IF Main.Errors.InMoldDryingErrors.TopMoldB.HeatingZone[2].PT100_TemperatureAboveMaximum THEN 
Topmold_B_heating_zone_2_temperature_above_250_degree_heating_element_switched_off.Raise(Main.timestampNanoseconds); 
END_IF 

IF Main.Errors.InMoldDryingErrors.TopMoldB.HeatingZone[2].PT100_TemperatureTooHighWarn THEN 
Topmold_B_heating_zone_2_temperature_above_230_degree.Raise(Main.timestampNanoseconds); 
END_IF 

IF Main.Errors.InMoldDryingErrors.TopMoldB.HeatingZone[3].PT100_ConnectorNotConnected THEN 
Topmold_B_heating_Zone_3_connector_not_connected.Raise(Main.timestampNanoseconds); 
END_IF 

IF Main.Errors.InMoldDryingErrors.TopMoldB.HeatingZone[3].PT100_HasWrongPosition THEN 
Topmold_B_heating_Zone_3_PT100_wrong_position.Raise(Main.timestampNanoseconds); 
END_IF 

IF Main.Errors.InMoldDryingErrors.TopMoldB.HeatingZone[3].PT100_Loose THEN 
Topmold_B_heating_Zone_3_PT100_loose.Raise(Main.timestampNanoseconds); 
END_IF 

IF Main.Errors.InMoldDryingErrors.TopMoldB.HeatingZone[3].PT100_NotInserted THEN 
Topmold_B_heating_Zone_3_PT100_not_inserted.Raise(Main.timestampNanoseconds); 
END_IF 

IF Main.Errors.InMoldDryingErrors.TopMoldB.HeatingZone[3].PT100_TempAboveSetpoint THEN 
Topmold_B_heating_Zone_3_Temperature_above_setpoint.Raise(Main.timestampNanoseconds); 
END_IF 

IF Main.Errors.InMoldDryingErrors.TopMoldB.HeatingZone[3].PT100_TempBelowSetpoint THEN 
Topmold_B_heating_Zone_3_Temperature_below_setpoint.Raise(Main.timestampNanoseconds); 
END_IF 

IF Main.Errors.InMoldDryingErrors.TopMoldB.HeatingZone[3].PT100_WireBreak THEN 
Topmold_B_heating_Zone_3_PT100_wirebreak.Raise(Main.timestampNanoseconds); 
END_IF 

IF Main.Errors.InMoldDryingErrors.TopMoldB.HeatingZone[3].Thermal THEN 
Topmold_B_heating_Zone_3_Thermal.Raise(Main.timestampNanoseconds); 
END_IF 

IF Main.Errors.InMoldDryingErrors.TopMoldB.HeatingZone[3].PT100_TemperatureAboveMaximum THEN 
Topmold_B_heating_zone_3_temperature_above_250_degree_heating_element_switched_off.Raise(Main.timestampNanoseconds); 
END_IF 

IF Main.Errors.InMoldDryingErrors.TopMoldB.HeatingZone[3].PT100_TemperatureTooHighWarn THEN 
Topmold_B_heating_zone_3_temperature_above_230_degree.Raise(Main.timestampNanoseconds); 
END_IF 

IF Main.Errors.InMoldDryingErrors.TopMoldB.HeatingZone[4].PT100_ConnectorNotConnected THEN 
Topmold_B_heating_Zone_4_connector_not_connected.Raise(Main.timestampNanoseconds); 
END_IF 

IF Main.Errors.InMoldDryingErrors.TopMoldB.HeatingZone[4].PT100_HasWrongPosition THEN 
Topmold_B_heating_Zone_4_PT100_wrong_position.Raise(Main.timestampNanoseconds); 
END_IF 

IF Main.Errors.InMoldDryingErrors.TopMoldB.HeatingZone[4].PT100_Loose THEN 
Topmold_B_heating_Zone_4_PT100_loose.Raise(Main.timestampNanoseconds); 
END_IF 

IF Main.Errors.InMoldDryingErrors.TopMoldB.HeatingZone[4].PT100_NotInserted THEN 
Topmold_B_heating_Zone_4_PT100_not_inserted.Raise(Main.timestampNanoseconds); 
END_IF 

IF Main.Errors.InMoldDryingErrors.TopMoldB.HeatingZone[4].PT100_TempAboveSetpoint THEN 
Topmold_B_heating_Zone_4_Temperature_above_setpoint.Raise(Main.timestampNanoseconds); 
END_IF 

IF Main.Errors.InMoldDryingErrors.TopMoldB.HeatingZone[4].PT100_TempBelowSetpoint THEN 
Topmold_B_heating_Zone_4_Temperature_below_setpoint.Raise(Main.timestampNanoseconds); 
END_IF 

IF Main.Errors.InMoldDryingErrors.TopMoldB.HeatingZone[4].PT100_WireBreak THEN 
Topmold_B_heating_Zone_4_PT100_wirebreak.Raise(Main.timestampNanoseconds); 
END_IF 

IF Main.Errors.InMoldDryingErrors.TopMoldB.HeatingZone[4].Thermal THEN 
Topmold_B_heating_Zone_4_Thermal.Raise(Main.timestampNanoseconds); 
END_IF 

IF Main.Errors.InMoldDryingErrors.TopMoldB.HeatingZone[4].PT100_TemperatureAboveMaximum THEN 
Topmold_B_heating_zone_4_temperature_above_250_degree_heating_element_switched_off.Raise(Main.timestampNanoseconds); 
END_IF 

IF Main.Errors.InMoldDryingErrors.TopMoldB.HeatingZone[4].PT100_TemperatureTooHighWarn THEN 
Topmold_B_heating_zone_4_temperature_above_230_degree.Raise(Main.timestampNanoseconds); 
END_IF 

IF Main.Errors.InMoldDryingErrors.TopMoldB.HeatingZone[5].PT100_ConnectorNotConnected THEN 
Topmold_B_heating_Zone_5_connector_not_connected.Raise(Main.timestampNanoseconds); 
END_IF 

IF Main.Errors.InMoldDryingErrors.TopMoldB.HeatingZone[5].PT100_HasWrongPosition THEN 
Topmold_B_heating_Zone_5_PT100_wrong_position.Raise(Main.timestampNanoseconds); 
END_IF 

IF Main.Errors.InMoldDryingErrors.TopMoldB.HeatingZone[5].PT100_Loose THEN 
Topmold_B_heating_Zone_5_PT100_loose.Raise(Main.timestampNanoseconds); 
END_IF 

IF Main.Errors.InMoldDryingErrors.TopMoldB.HeatingZone[5].PT100_NotInserted THEN 
Topmold_B_heating_Zone_5_PT100_not_inserted.Raise(Main.timestampNanoseconds); 
END_IF 

IF Main.Errors.InMoldDryingErrors.TopMoldB.HeatingZone[5].PT100_TempAboveSetpoint THEN 
Topmold_B_heating_Zone_5_Temperature_above_setpoint.Raise(Main.timestampNanoseconds); 
END_IF 

IF Main.Errors.InMoldDryingErrors.TopMoldB.HeatingZone[5].PT100_TempBelowSetpoint THEN 
Topmold_B_heating_Zone_5_Temperature_below_setpoint.Raise(Main.timestampNanoseconds); 
END_IF 

IF Main.Errors.InMoldDryingErrors.TopMoldB.HeatingZone[5].PT100_WireBreak THEN 
Topmold_B_heating_Zone_5_PT100_wirebreak.Raise(Main.timestampNanoseconds); 
END_IF 

IF Main.Errors.InMoldDryingErrors.TopMoldB.HeatingZone[5].Thermal THEN 
Topmold_B_heating_Zone_5_Thermal.Raise(Main.timestampNanoseconds); 
END_IF 

IF Main.Errors.InMoldDryingErrors.TopMoldB.HeatingZone[5].PT100_TemperatureAboveMaximum THEN 
Topmold_B_heating_zone_5_temperature_above_250_degree_heating_element_switched_off.Raise(Main.timestampNanoseconds); 
END_IF 

IF Main.Errors.InMoldDryingErrors.TopMoldB.HeatingZone[5].PT100_TemperatureTooHighWarn THEN 
Topmold_B_heating_zone_5_temperature_above_230_degree.Raise(Main.timestampNanoseconds); 
END_IF 

IF Main.Errors.InMoldDryingErrors.TopMoldB.HeatingZone[6].PT100_ConnectorNotConnected THEN 
Topmold_B_heating_Zone_6_connector_not_connected.Raise(Main.timestampNanoseconds); 
END_IF 

IF Main.Errors.InMoldDryingErrors.TopMoldB.HeatingZone[6].PT100_HasWrongPosition THEN 
Topmold_B_heating_Zone_6_PT100_wrong_position.Raise(Main.timestampNanoseconds); 
END_IF 

IF Main.Errors.InMoldDryingErrors.TopMoldB.HeatingZone[6].PT100_Loose THEN 
Topmold_B_heating_Zone_6_PT100_loose.Raise(Main.timestampNanoseconds); 
END_IF 

IF Main.Errors.InMoldDryingErrors.TopMoldB.HeatingZone[6].PT100_NotInserted THEN 
Topmold_B_heating_Zone_6_PT100_not_inserted.Raise(Main.timestampNanoseconds); 
END_IF 

IF Main.Errors.InMoldDryingErrors.TopMoldB.HeatingZone[6].PT100_TempAboveSetpoint THEN 
Topmold_B_heating_Zone_6_Temperature_above_setpoint.Raise(Main.timestampNanoseconds); 
END_IF 

IF Main.Errors.InMoldDryingErrors.TopMoldB.HeatingZone[6].PT100_TempBelowSetpoint THEN 
Topmold_B_heating_Zone_6_Temperature_below_setpoint.Raise(Main.timestampNanoseconds); 
END_IF 

IF Main.Errors.InMoldDryingErrors.TopMoldB.HeatingZone[6].PT100_WireBreak THEN 
Topmold_B_heating_Zone_6_PT100_wirebreak.Raise(Main.timestampNanoseconds); 
END_IF 

IF Main.Errors.InMoldDryingErrors.TopMoldB.HeatingZone[6].Thermal THEN 
Topmold_B_heating_Zone_6_Thermal.Raise(Main.timestampNanoseconds); 
END_IF 

IF Main.Errors.InMoldDryingErrors.TopMoldB.HeatingZone[6].PT100_TemperatureAboveMaximum THEN 
Topmold_B_heating_zone_6_temperature_above_250_degree_heating_element_switched_off.Raise(Main.timestampNanoseconds); 
END_IF 

IF Main.Errors.InMoldDryingErrors.TopMoldB.HeatingZone[6].PT100_TemperatureTooHighWarn THEN 
Topmold_B_heating_zone_6_temperature_above_230_degree.Raise(Main.timestampNanoseconds); 
END_IF 

IF Main.Errors.InMoldDryingErrors.TopMoldB.Hydraulic.BallufError THEN 
Bottom_mold_B_error_on_balluf.Raise(Main.timestampNanoseconds); 
END_IF 

IF Main.Errors.InMoldDryingErrors.TopMoldB.Hydraulic.IsMovingWithoutActivation THEN 
Bottom_mold_B_is_moving_without_activation.Raise(Main.timestampNanoseconds); 
END_IF 

IF FALSE THEN 
Top_mold_B_Bot_side_pressure_too_high.Raise(Main.timestampNanoseconds); 
END_IF 

IF FALSE THEN 
Top_mold_B_Rot_side_pressure_too_high.Raise(Main.timestampNanoseconds); 
END_IF 

IF Main.Errors.InMoldDryingErrors.BottomMoldB.HeatingZone[1].PT100_ConnectorNotConnected THEN 
Bottom_mold_B_heating_Zone_1_connector_not_connected.Raise(Main.timestampNanoseconds); 
END_IF 

IF Main.Errors.InMoldDryingErrors.BottomMoldB.HeatingZone[1].PT100_HasWrongPosition THEN 
Bottom_mold_B_heating_Zone_1_PT100_wrong_position.Raise(Main.timestampNanoseconds); 
END_IF 

IF Main.Errors.InMoldDryingErrors.BottomMoldB.HeatingZone[1].PT100_Loose THEN 
Bottom_mold_B_heating_Zone_1_PT100_loose.Raise(Main.timestampNanoseconds); 
END_IF 

IF Main.Errors.InMoldDryingErrors.BottomMoldB.HeatingZone[1].PT100_NotInserted THEN 
Bottom_mold_B_heating_Zone_1_PT100_not_inserted.Raise(Main.timestampNanoseconds); 
END_IF 

IF Main.Errors.InMoldDryingErrors.BottomMoldB.HeatingZone[1].PT100_TempAboveSetpoint THEN 
Bottom_mold_B_heating_Zone_1_Temperature_above_setpoint.Raise(Main.timestampNanoseconds); 
END_IF 

IF Main.Errors.InMoldDryingErrors.BottomMoldB.HeatingZone[1].PT100_TempBelowSetpoint THEN 
Bottom_mold_B_heating_Zone_1_Temperature_below_setpoint.Raise(Main.timestampNanoseconds); 
END_IF 

IF Main.Errors.InMoldDryingErrors.BottomMoldB.HeatingZone[1].PT100_WireBreak THEN 
Bottom_mold_B_heating_Zone_1_PT100_wirebreak.Raise(Main.timestampNanoseconds); 
END_IF 

IF Main.Errors.InMoldDryingErrors.BottomMoldB.HeatingZone[1].Thermal THEN 
Bottom_mold_B_heating_Zone_1_Thermal.Raise(Main.timestampNanoseconds); 
END_IF 

IF Main.Errors.InMoldDryingErrors.BottomMoldB.HeatingZone[1].PT100_TemperatureAboveMaximum THEN 
Bottom_mold_B_heating_zone_1_temperature_above_250_degree_heating_element_switched_off.Raise(Main.timestampNanoseconds); 
END_IF 

IF Main.Errors.InMoldDryingErrors.BottomMoldB.HeatingZone[1].PT100_TemperatureTooHighWarn THEN 
Bottom_mold_B_heating_zone_1_temperature_above_230_degree.Raise(Main.timestampNanoseconds); 
END_IF 

IF Main.Errors.InMoldDryingErrors.BottomMoldB.HeatingZone[2].PT100_ConnectorNotConnected THEN 
Bottom_mold_B_heating_Zone_2_connector_not_connected.Raise(Main.timestampNanoseconds); 
END_IF 

IF Main.Errors.InMoldDryingErrors.BottomMoldB.HeatingZone[2].PT100_HasWrongPosition THEN 
Bottom_mold_B_heating_Zone_2_PT100_wrong_position.Raise(Main.timestampNanoseconds); 
END_IF 

IF Main.Errors.InMoldDryingErrors.BottomMoldB.HeatingZone[2].PT100_Loose THEN 
Bottom_mold_B_heating_Zone_2_PT100_loose.Raise(Main.timestampNanoseconds); 
END_IF 

IF Main.Errors.InMoldDryingErrors.BottomMoldB.HeatingZone[2].PT100_NotInserted THEN 
Bottom_mold_B_heating_Zone_2_PT100_not_inserted.Raise(Main.timestampNanoseconds); 
END_IF 

IF Main.Errors.InMoldDryingErrors.BottomMoldB.HeatingZone[2].PT100_TempAboveSetpoint THEN 
Bottom_mold_B_heating_Zone_2_Temperature_above_setpoint.Raise(Main.timestampNanoseconds); 
END_IF 

IF Main.Errors.InMoldDryingErrors.BottomMoldB.HeatingZone[2].PT100_TempBelowSetpoint THEN 
Bottom_mold_B_heating_Zone_2_Temperature_below_setpoint.Raise(Main.timestampNanoseconds); 
END_IF 

IF Main.Errors.InMoldDryingErrors.BottomMoldB.HeatingZone[2].PT100_WireBreak THEN 
Bottom_mold_B_heating_Zone_2_PT100_wirebreak.Raise(Main.timestampNanoseconds); 
END_IF 

IF Main.Errors.InMoldDryingErrors.BottomMoldB.HeatingZone[2].Thermal THEN 
Bottom_mold_B_heating_Zone_2_Thermal.Raise(Main.timestampNanoseconds); 
END_IF 

IF Main.Errors.InMoldDryingErrors.BottomMoldB.HeatingZone[2].PT100_TemperatureAboveMaximum THEN 
Bottom_mold_B_heating_zone_2_temperature_above_250_degree_heating_element_switched_off.Raise(Main.timestampNanoseconds); 
END_IF 

IF Main.Errors.InMoldDryingErrors.BottomMoldB.HeatingZone[2].PT100_TemperatureTooHighWarn THEN 
Bottom_mold_B_heating_zone_2_temperature_above_230_degree.Raise(Main.timestampNanoseconds); 
END_IF 

IF Main.Errors.InMoldDryingErrors.BottomMoldB.HeatingZone[3].PT100_ConnectorNotConnected THEN 
Bottom_mold_B_heating_Zone_3_connector_not_connected.Raise(Main.timestampNanoseconds); 
END_IF 

IF Main.Errors.InMoldDryingErrors.BottomMoldB.HeatingZone[3].PT100_HasWrongPosition THEN 
Bottom_mold_B_heating_Zone_3_PT100_wrong_position.Raise(Main.timestampNanoseconds); 
END_IF 

IF Main.Errors.InMoldDryingErrors.BottomMoldB.HeatingZone[3].PT100_Loose THEN 
Bottom_mold_B_heating_Zone_3_PT100_loose.Raise(Main.timestampNanoseconds); 
END_IF 

IF Main.Errors.InMoldDryingErrors.BottomMoldB.HeatingZone[3].PT100_NotInserted THEN 
Bottom_mold_B_heating_Zone_3_PT100_not_inserted.Raise(Main.timestampNanoseconds); 
END_IF 

IF Main.Errors.InMoldDryingErrors.BottomMoldB.HeatingZone[3].PT100_TempAboveSetpoint THEN 
Bottom_mold_B_heating_Zone_3_Temperature_above_setpoint.Raise(Main.timestampNanoseconds); 
END_IF 

IF Main.Errors.InMoldDryingErrors.BottomMoldB.HeatingZone[3].PT100_TempBelowSetpoint THEN 
Bottom_mold_B_heating_Zone_3_Temperature_below_setpoint.Raise(Main.timestampNanoseconds); 
END_IF 

IF Main.Errors.InMoldDryingErrors.BottomMoldB.HeatingZone[3].PT100_WireBreak THEN 
Bottom_mold_B_heating_Zone_3_PT100_wirebreak.Raise(Main.timestampNanoseconds); 
END_IF 

IF Main.Errors.InMoldDryingErrors.BottomMoldB.HeatingZone[3].Thermal THEN 
Bottom_mold_B_heating_Zone_3_Thermal.Raise(Main.timestampNanoseconds); 
END_IF 

IF Main.Errors.InMoldDryingErrors.BottomMoldB.HeatingZone[3].PT100_TemperatureAboveMaximum THEN 
Bottom_mold_B_heating_zone_3_temperature_above_250_degree_heating_element_switched_off.Raise(Main.timestampNanoseconds); 
END_IF 

IF Main.Errors.InMoldDryingErrors.BottomMoldB.HeatingZone[3].PT100_TemperatureTooHighWarn THEN 
Bottom_mold_B_heating_zone_3_temperature_above_230_degree.Raise(Main.timestampNanoseconds); 
END_IF 

IF Main.Errors.InMoldDryingErrors.BottomMoldB.HeatingZone[4].PT100_ConnectorNotConnected THEN 
Bottom_mold_B_heating_Zone_4_connector_not_connected.Raise(Main.timestampNanoseconds); 
END_IF 

IF Main.Errors.InMoldDryingErrors.BottomMoldB.HeatingZone[4].PT100_HasWrongPosition THEN 
Bottom_mold_B_heating_Zone_4_PT100_wrong_position.Raise(Main.timestampNanoseconds); 
END_IF 

IF Main.Errors.InMoldDryingErrors.BottomMoldB.HeatingZone[4].PT100_Loose THEN 
Bottom_mold_B_heating_Zone_4_PT100_loose.Raise(Main.timestampNanoseconds); 
END_IF 

IF Main.Errors.InMoldDryingErrors.BottomMoldB.HeatingZone[4].PT100_NotInserted THEN 
Bottom_mold_B_heating_Zone_4_PT100_not_inserted.Raise(Main.timestampNanoseconds); 
END_IF 

IF Main.Errors.InMoldDryingErrors.BottomMoldB.HeatingZone[4].PT100_TempAboveSetpoint THEN 
Bottom_mold_B_heating_Zone_4_Temperature_above_setpoint.Raise(Main.timestampNanoseconds); 
END_IF 

IF Main.Errors.InMoldDryingErrors.BottomMoldB.HeatingZone[4].PT100_TempBelowSetpoint THEN 
Bottom_mold_B_heating_Zone_4_Temperature_below_setpoint.Raise(Main.timestampNanoseconds); 
END_IF 

IF Main.Errors.InMoldDryingErrors.BottomMoldB.HeatingZone[4].PT100_WireBreak THEN 
Bottom_mold_B_heating_Zone_4_PT100_wirebreak.Raise(Main.timestampNanoseconds); 
END_IF 

IF Main.Errors.InMoldDryingErrors.BottomMoldB.HeatingZone[4].Thermal THEN 
Bottom_mold_B_heating_Zone_4_Thermal.Raise(Main.timestampNanoseconds); 
END_IF 

IF Main.Errors.InMoldDryingErrors.BottomMoldB.HeatingZone[4].PT100_TemperatureAboveMaximum THEN 
Bottom_mold_B_heating_zone_4_temperature_above_250_degree_heating_element_switched_off.Raise(Main.timestampNanoseconds); 
END_IF 

IF Main.Errors.InMoldDryingErrors.BottomMoldB.HeatingZone[4].PT100_TemperatureTooHighWarn THEN 
Bottom_mold_B_heating_zone_4_temperature_above_230_degree.Raise(Main.timestampNanoseconds); 
END_IF 

IF Main.Errors.InMoldDryingErrors.BottomMoldB.HeatingZone[5].PT100_ConnectorNotConnected THEN 
Bottom_mold_B_heating_Zone_5_connector_not_connected.Raise(Main.timestampNanoseconds); 
END_IF 

IF Main.Errors.InMoldDryingErrors.BottomMoldB.HeatingZone[5].PT100_HasWrongPosition THEN 
Bottom_mold_B_heating_Zone_5_PT100_wrong_position.Raise(Main.timestampNanoseconds); 
END_IF 

IF Main.Errors.InMoldDryingErrors.BottomMoldB.HeatingZone[5].PT100_Loose THEN 
Bottom_mold_B_heating_Zone_5_PT100_loose.Raise(Main.timestampNanoseconds); 
END_IF 

IF Main.Errors.InMoldDryingErrors.BottomMoldB.HeatingZone[5].PT100_NotInserted THEN 
Bottom_mold_B_heating_Zone_5_PT100_not_inserted.Raise(Main.timestampNanoseconds); 
END_IF 

IF Main.Errors.InMoldDryingErrors.BottomMoldB.HeatingZone[5].PT100_TempAboveSetpoint THEN 
Bottom_mold_B_heating_Zone_5_Temperature_above_setpoint.Raise(Main.timestampNanoseconds); 
END_IF 

IF Main.Errors.InMoldDryingErrors.BottomMoldB.HeatingZone[5].PT100_TempBelowSetpoint THEN 
Bottom_mold_B_heating_Zone_5_Temperature_below_setpoint.Raise(Main.timestampNanoseconds); 
END_IF 

IF Main.Errors.InMoldDryingErrors.BottomMoldB.HeatingZone[5].PT100_WireBreak THEN 
Bottom_mold_B_heating_Zone_5_PT100_wirebreak.Raise(Main.timestampNanoseconds); 
END_IF 

IF Main.Errors.InMoldDryingErrors.BottomMoldB.HeatingZone[5].Thermal THEN 
Bottom_mold_B_heating_Zone_5_Thermal.Raise(Main.timestampNanoseconds); 
END_IF 

IF Main.Errors.InMoldDryingErrors.BottomMoldB.HeatingZone[5].PT100_TemperatureAboveMaximum THEN 
Bottom_mold_B_heating_zone_5_temperature_above_250_degree_heating_element_switched_off.Raise(Main.timestampNanoseconds); 
END_IF 

IF Main.Errors.InMoldDryingErrors.BottomMoldB.HeatingZone[5].PT100_TemperatureTooHighWarn THEN 
Bottom_mold_B_heating_zone_5_temperature_above_230_degree.Raise(Main.timestampNanoseconds); 
END_IF 

IF Main.Errors.InMoldDryingErrors.BottomMoldB.HeatingZone[6].PT100_ConnectorNotConnected THEN 
Bottom_mold_B_heating_Zone_6_connector_not_connected.Raise(Main.timestampNanoseconds); 
END_IF 

IF Main.Errors.InMoldDryingErrors.BottomMoldB.HeatingZone[6].PT100_HasWrongPosition THEN 
Bottom_mold_B_heating_Zone_6_PT100_wrong_position.Raise(Main.timestampNanoseconds); 
END_IF 

IF Main.Errors.InMoldDryingErrors.BottomMoldB.HeatingZone[6].PT100_Loose THEN 
Bottom_mold_B_heating_Zone_6_PT100_loose.Raise(Main.timestampNanoseconds); 
END_IF 

IF Main.Errors.InMoldDryingErrors.BottomMoldB.HeatingZone[6].PT100_NotInserted THEN 
Bottom_mold_B_heating_Zone_6_PT100_not_inserted.Raise(Main.timestampNanoseconds); 
END_IF 

IF Main.Errors.InMoldDryingErrors.BottomMoldB.HeatingZone[6].PT100_TempAboveSetpoint THEN 
Bottom_mold_B_heating_Zone_6_Temperature_above_setpoint.Raise(Main.timestampNanoseconds); 
END_IF 

IF Main.Errors.InMoldDryingErrors.BottomMoldB.HeatingZone[6].PT100_TempBelowSetpoint THEN 
Bottom_mold_B_heating_Zone_6_Temperature_below_setpoint.Raise(Main.timestampNanoseconds); 
END_IF 

IF Main.Errors.InMoldDryingErrors.BottomMoldB.HeatingZone[6].PT100_WireBreak THEN 
Bottom_mold_B_heating_Zone_6_PT100_wirebreak.Raise(Main.timestampNanoseconds); 
END_IF 

IF Main.Errors.InMoldDryingErrors.BottomMoldB.HeatingZone[6].Thermal THEN 
Bottom_mold_B_heating_Zone_6_Thermal.Raise(Main.timestampNanoseconds); 
END_IF 

IF Main.Errors.InMoldDryingErrors.BottomMoldB.HeatingZone[6].PT100_TemperatureAboveMaximum THEN 
Bottom_mold_B_heating_zone_6_temperature_above_250_degree_heating_element_switched_off.Raise(Main.timestampNanoseconds); 
END_IF 

IF Main.Errors.InMoldDryingErrors.BottomMoldB.HeatingZone[6].PT100_TemperatureTooHighWarn THEN 
Bottom_mold_B_heating_zone_6_temperature_above_230_degree.Raise(Main.timestampNanoseconds); 
END_IF 

IF Main.Errors.InMoldDryingErrors.BottomMoldA.HorizontalCilinder.Cilinder THEN 
Takeout_unit_A_horizontal_cylinder_error.Raise(Main.timestampNanoseconds); 
END_IF 

IF Main.Errors.InMoldDryingErrors.BottomMoldA.HorizontalCilinder.CilinderSlow_IN THEN 
Takeout_unit_A_horizontal_cylinder_timeout_in.Raise(Main.timestampNanoseconds); 
END_IF 

IF Main.Errors.InMoldDryingErrors.BottomMoldA.HorizontalCilinder.CilinderSlow_OUT THEN 
Takeout_unit_A_horizontal_cylinder_timeout_out.Raise(Main.timestampNanoseconds); 
END_IF 

IF Main.Errors.InMoldDryingErrors.BottomMoldB.HorizontalCilinder.Cilinder THEN 
Takeout_unit_B_horizontal_cylinder_error.Raise(Main.timestampNanoseconds); 
END_IF 

IF Main.Errors.InMoldDryingErrors.BottomMoldB.HorizontalCilinder.CilinderSlow_IN THEN 
Takeout_unit_B_horizontal_cylinder_timeout_in.Raise(Main.timestampNanoseconds); 
END_IF 

IF Main.Errors.InMoldDryingErrors.BottomMoldB.HorizontalCilinder.CilinderSlow_OUT THEN 
Takeout_unit_B_horizontal_cylinder_timeout_out.Raise(Main.timestampNanoseconds); 
END_IF 

IF Main.Errors.InMoldDryingErrors.BottomMoldA.VerticalCilinder.Cilinder THEN 
Takeout_unit_A_vertical_cylinder_error.Raise(Main.timestampNanoseconds); 
END_IF 

IF Main.Errors.InMoldDryingErrors.BottomMoldA.VerticalCilinder.CilinderSlow_IN THEN 
Takeout_unit_A_vertical_cylinder_timeout_in.Raise(Main.timestampNanoseconds); 
END_IF 

IF Main.Errors.InMoldDryingErrors.BottomMoldA.VerticalCilinder.CilinderSlow_OUT THEN 
Takeout_unit_A_vertical_cylinder_timeout_out.Raise(Main.timestampNanoseconds); 
END_IF 

IF Main.Errors.InMoldDryingErrors.BottomMoldB.VerticalCilinder.Cilinder THEN 
Takeout_unit_B_vertical_cylinder_error.Raise(Main.timestampNanoseconds); 
END_IF 

IF Main.Errors.InMoldDryingErrors.BottomMoldB.VerticalCilinder.CilinderSlow_IN THEN 
Takeout_unit_B_vertical_cylinder_timeout_in.Raise(Main.timestampNanoseconds); 
END_IF 

IF Main.Errors.InMoldDryingErrors.BottomMoldB.VerticalCilinder.CilinderSlow_OUT THEN 
Takeout_unit_B_vertical_cylinder_timeout_out.Raise(Main.timestampNanoseconds); 
END_IF 

IF Main.Errors.InMoldDryingErrors.BottomMoldA.VacuumSection[1] THEN 
Takeout_unit_A_error_on_vacuum_section_1.Raise(Main.timestampNanoseconds); 
END_IF 

IF Main.Errors.InMoldDryingErrors.BottomMoldA.VacuumSection[2] THEN 
Takeout_unit_A_error_on_vacuum_section_2.Raise(Main.timestampNanoseconds); 
END_IF 

IF Main.Errors.InMoldDryingErrors.BottomMoldA.VacuumSection[3] THEN 
Takeout_unit_A_error_on_vacuum_section_3.Raise(Main.timestampNanoseconds); 
END_IF 

IF Main.Errors.InMoldDryingErrors.BottomMoldA.VacuumSection[4] THEN 
Takeout_unit_A_error_on_vacuum_section_4.Raise(Main.timestampNanoseconds); 
END_IF 

IF Main.Errors.InMoldDryingErrors.BottomMoldB.VacuumSection[1] THEN 
Takeout_unit_B_error_on_vacuum_section_1.Raise(Main.timestampNanoseconds); 
END_IF 

IF Main.Errors.InMoldDryingErrors.BottomMoldB.VacuumSection[2] THEN 
Takeout_unit_B_error_on_vacuum_section_2.Raise(Main.timestampNanoseconds); 
END_IF 

IF Main.Errors.InMoldDryingErrors.BottomMoldB.VacuumSection[3] THEN 
Takeout_unit_B_error_on_vacuum_section_3.Raise(Main.timestampNanoseconds); 
END_IF 

IF Main.Errors.InMoldDryingErrors.BottomMoldB.VacuumSection[4] THEN 
Takeout_unit_B_error_on_vacuum_section_4.Raise(Main.timestampNanoseconds); 
END_IF 

IF Main.Errors.InMoldDryingErrors.ProductForming.HydraulicPump.Maintenance THEN 
Machine_pond_hydraulic_pump_maintenance_switch.Raise(Main.timestampNanoseconds); 
END_IF 

IF Main.Errors.InMoldDryingErrors.ProductForming.HydraulicPump.Thermal THEN 
Machine_pond_hydraulic_pump_thermal_error.Raise(Main.timestampNanoseconds); 
END_IF 

IF Main.Errors.InMoldDryingErrors.ProductForming.MachinePond.FeedingPulp.Cilinder THEN 
Machine_oond_pulp_feeding_cylinder_error.Raise(Main.timestampNanoseconds); 
END_IF 

IF Main.Errors.InMoldDryingErrors.ProductForming.MachinePond.FeedingPulp.CilinderSlow_IN THEN 
Machine_pond_pulp_feeding_cylinder_timeout_in.Raise(Main.timestampNanoseconds); 
END_IF 

IF Main.Errors.InMoldDryingErrors.ProductForming.MachinePond.FeedingPulp.CilinderSlow_OUT THEN 
Machine_pond_pulp_feeding_cylinder_timeout_out.Raise(Main.timestampNanoseconds); 
END_IF 

IF Main.Errors.InMoldDryingErrors.TransferMold.HydraulicCilinder.BallufError THEN 
Transfermold_error_on_balluf.Raise(Main.timestampNanoseconds); 
END_IF 

IF Main.Errors.InMoldDryingErrors.TransferMold.HydraulicCilinder.IsMovingWithoutActivation THEN 
Transfermold_is_moving_without_activation.Raise(Main.timestampNanoseconds); 
END_IF 

IF Main.Errors.InMoldDryingErrors.RH_BotMoldAToCoolForTrMDown THEN 
RHSR_Bottommold_A_too_cool_for_transfermold_to_come_down.Raise(Main.timestampNanoseconds); 
END_IF 

IF Main.Errors.InMoldDryingErrors.RH_BotMoldBToCoolForTrMDown THEN 
RHSR_Bottommold_B_too_cool_for_transfermold_to_come_down.Raise(Main.timestampNanoseconds); 
END_IF 

IF Main.Errors.ProductHandlingErrors.Gantry_A.Collision THEN 
Gantry_A_collision_detected.Raise(Main.timestampNanoseconds); 
END_IF 

IF Main.Errors.ProductHandlingErrors.Gantry_A.EndLimitHorBack THEN 
Gantry_A_Horizontal_limit_endswitch_backside.Raise(Main.timestampNanoseconds); 
END_IF 

IF Main.Errors.ProductHandlingErrors.Gantry_A.EndLimitHorFront THEN 
Gantry_A_Horizontal_limit_endswitch_frontside.Raise(Main.timestampNanoseconds); 
END_IF 

IF Main.Errors.ProductHandlingErrors.Gantry_A.EndLimitVertDown THEN 
Gantry_A_vertical_limit_endswitch_down.Raise(Main.timestampNanoseconds); 
END_IF 

IF Main.Errors.ProductHandlingErrors.Gantry_A.EndLimitVertUp THEN 
Gantry_A_vertical_limit_endswitch_up.Raise(Main.timestampNanoseconds); 
END_IF 

IF Main.Errors.ProductHandlingErrors.Gantry_A.HorizontalNCAxisError.exDriveAbsoluut THEN 
Gantry_A_Horizontal_Drive_absoluut_error.Raise(Main.timestampNanoseconds); 
END_IF 

IF Main.Errors.ProductHandlingErrors.Gantry_A.HorizontalNCAxisError.exDriveJog THEN 
Gantry_A_Horizontal_Drive_Jog_error.Raise(Main.timestampNanoseconds); 
END_IF 

IF Main.Errors.ProductHandlingErrors.Gantry_A.HorizontalNCAxisError.exDrivePower THEN 
Gantry_A_Horizontal_Drive_power_error.Raise(Main.timestampNanoseconds); 
END_IF 

IF Main.Errors.ProductHandlingErrors.Gantry_A.HorizontalNCAxisError.exDriveReset THEN 
Gantry_A_Horizontal_Drive_reset.Raise(Main.timestampNanoseconds); 
END_IF 

IF Main.Errors.ProductHandlingErrors.Gantry_A.HorizontalNCAxisError.exDriveStatus THEN 
Gantry_A_Horizontal_Drive_status.Raise(Main.timestampNanoseconds); 
END_IF 

IF Main.Errors.ProductHandlingErrors.Gantry_A.HorizontalNCAxisError.exDriveStop THEN 
Gantry_A_Horizontal_Drive_stop_error.Raise(Main.timestampNanoseconds); 
END_IF 

IF Main.Errors.ProductHandlingErrors.Gantry_A.HorizontalNCAxisError.exDriveVelocity THEN 
Gantry_A_Horizontal_Drive_velocity_error.Raise(Main.timestampNanoseconds); 
END_IF 

IF Main.Errors.ProductHandlingErrors.Gantry_A.HorizontalNCAxisError.exHome THEN 
Gantry_A_Horizontal_Drive_home_error.Raise(Main.timestampNanoseconds); 
END_IF 

IF Main.Errors.ProductHandlingErrors.Gantry_A.HorizontalNCAxisError.exLagError THEN 
Gantry_A_Horizontal_Drive_lag_error.Raise(Main.timestampNanoseconds); 
END_IF 

IF Main.Errors.ProductHandlingErrors.Gantry_A.HorizontalNCAxisError.exReadParameter THEN 
Gantry_A_Horizontal_Drive_read_parameter_error.Raise(Main.timestampNanoseconds); 
END_IF 

IF Main.Errors.ProductHandlingErrors.Gantry_A.HorizontalNCAxisError.exWriteParameter THEN 
Gantry_A_Horizontal_Drive_write_parameter_error.Raise(Main.timestampNanoseconds); 
END_IF 

IF Main.Errors.ProductHandlingErrors.Gantry_B.Collision THEN 
Gantry_B_collision_detected.Raise(Main.timestampNanoseconds); 
END_IF 

IF Main.Errors.ProductHandlingErrors.Gantry_B.EndLimitHorBack THEN 
Gantry_B_horizontal_limit_endswitch_backside.Raise(Main.timestampNanoseconds); 
END_IF 

IF Main.Errors.ProductHandlingErrors.Gantry_B.EndLimitHorFront THEN 
Gantry_B_horizontal_limit_endswitch_frontside.Raise(Main.timestampNanoseconds); 
END_IF 

IF Main.Errors.ProductHandlingErrors.Gantry_B.EndLimitVertDown THEN 
Gantry_B_vertical_limit_endswitch_down.Raise(Main.timestampNanoseconds); 
END_IF 

IF Main.Errors.ProductHandlingErrors.Gantry_B.EndLimitVertUp THEN 
Gantry_B_vertical_limit_endswitch_up.Raise(Main.timestampNanoseconds); 
END_IF 

IF Main.Errors.ProductHandlingErrors.Gantry_B.HorizontalNCAxisError.exDriveAbsoluut THEN 
Gantry_B_Horizontal_Drive_absoluut_error.Raise(Main.timestampNanoseconds); 
END_IF 

IF Main.Errors.ProductHandlingErrors.Gantry_B.HorizontalNCAxisError.exDriveJog THEN 
Gantry_B_Horizontal_Drive_Jog_error.Raise(Main.timestampNanoseconds); 
END_IF 

IF Main.Errors.ProductHandlingErrors.Gantry_B.HorizontalNCAxisError.exDrivePower THEN 
Gantry_B_Horizontal_Drive_power_error.Raise(Main.timestampNanoseconds); 
END_IF 

IF Main.Errors.ProductHandlingErrors.Gantry_B.HorizontalNCAxisError.exDriveReset THEN 
Gantry_B_Horizontal_Drive_reset.Raise(Main.timestampNanoseconds); 
END_IF 

IF Main.Errors.ProductHandlingErrors.Gantry_B.HorizontalNCAxisError.exDriveStatus THEN 
Gantry_B_Horizontal_Drive_status.Raise(Main.timestampNanoseconds); 
END_IF 

IF Main.Errors.ProductHandlingErrors.Gantry_B.HorizontalNCAxisError.exDriveStop THEN 
Gantry_B_Horizontal_Drive_stop_error.Raise(Main.timestampNanoseconds); 
END_IF 

IF Main.Errors.ProductHandlingErrors.Gantry_B.HorizontalNCAxisError.exDriveVelocity THEN 
Gantry_B_Horizontal_Drive_velocity_error.Raise(Main.timestampNanoseconds); 
END_IF 

IF Main.Errors.ProductHandlingErrors.Gantry_B.HorizontalNCAxisError.exHome THEN 
Gantry_B_Horizontal_Drive_home_error.Raise(Main.timestampNanoseconds); 
END_IF 

IF Main.Errors.ProductHandlingErrors.Gantry_B.HorizontalNCAxisError.exLagError THEN 
Gantry_B_Horizontal_Drive_lag_error.Raise(Main.timestampNanoseconds); 
END_IF 

IF Main.Errors.ProductHandlingErrors.Gantry_B.HorizontalNCAxisError.exReadParameter THEN 
Gantry_B_Horizontal_Drive_read_parameter_error.Raise(Main.timestampNanoseconds); 
END_IF 

IF Main.Errors.ProductHandlingErrors.Gantry_B.HorizontalNCAxisError.exWriteParameter THEN 
Gantry_B_Horizontal_Drive_write_parameter_error.Raise(Main.timestampNanoseconds); 
END_IF 

IF Main.Errors.ProductHandlingErrors.RH_HorMovingVertNotAtTranspPos_A THEN 
RHSR_product_handling_gantry_A_is_moving_horizotal_while_vertical_not_on_position.Raise(Main.timestampNanoseconds); 
END_IF 

IF Main.Errors.ProductHandlingErrors.RH_HorMovingVertNotAtTranspPos_B THEN 
RHSR_product_handling_gantry_B_is_moving_horizotal_while_vertical_not_on_position.Raise(Main.timestampNanoseconds); 
END_IF 

IF Main.Errors.ProductHandlingErrors.RH_VertMovingHorNotInPos_A THEN 
RHSR_product_handling_gantry_A_is_moving_vertical_while_horizontal_not_on_position.Raise(Main.timestampNanoseconds); 
END_IF 

IF Main.Errors.ProductHandlingErrors.RH_VertMovingHorNotInPos_B THEN 
RHSR_product_handling_gantry_B_is_moving_vertical_while_horizontal_not_on_position.Raise(Main.timestampNanoseconds); 
END_IF 

IF Main.Errors.InMoldDryingErrors.ProductForming.SprayBar.NCAxisError.exDriveAbsoluut THEN 
Spraybar_Drive_absoluut_error.Raise(Main.timestampNanoseconds); 
END_IF 

IF Main.Errors.InMoldDryingErrors.ProductForming.SprayBar.NCAxisError.exDriveJog THEN 
Spraybar_Drive_Jog_error.Raise(Main.timestampNanoseconds); 
END_IF 

IF Main.Errors.InMoldDryingErrors.ProductForming.SprayBar.NCAxisError.exDrivePower THEN 
Spraybar_Drive_power_error.Raise(Main.timestampNanoseconds); 
END_IF 

IF Main.Errors.InMoldDryingErrors.ProductForming.SprayBar.NCAxisError.exDriveReset THEN 
Spraybar_Drive_reset.Raise(Main.timestampNanoseconds); 
END_IF 

IF Main.Errors.InMoldDryingErrors.ProductForming.SprayBar.NCAxisError.exDriveStatus THEN 
Spraybar_Drive_status.Raise(Main.timestampNanoseconds); 
END_IF 

IF Main.Errors.InMoldDryingErrors.ProductForming.SprayBar.NCAxisError.exDriveStop THEN 
Spraybar_Drive_stop_error.Raise(Main.timestampNanoseconds); 
END_IF 

IF Main.Errors.InMoldDryingErrors.ProductForming.SprayBar.NCAxisError.exDriveVelocity THEN 
Spraybar_Drive_velocity_error.Raise(Main.timestampNanoseconds); 
END_IF 

IF Main.Errors.InMoldDryingErrors.ProductForming.SprayBar.NCAxisError.exHome THEN 
Spraybar_Drive_home_error.Raise(Main.timestampNanoseconds); 
END_IF 

IF Main.Errors.InMoldDryingErrors.ProductForming.SprayBar.NCAxisError.exLagError THEN 
Spraybar_Drive_lag_error.Raise(Main.timestampNanoseconds); 
END_IF 

IF Main.Errors.InMoldDryingErrors.ProductForming.SprayBar.NCAxisError.exReadParameter THEN 
Spraybar_Drive_read_parameter_error.Raise(Main.timestampNanoseconds); 
END_IF 

IF Main.Errors.InMoldDryingErrors.ProductForming.SprayBar.NCAxisError.exWriteParameter THEN 
Spraybar_Drive_write_parameter_error.Raise(Main.timestampNanoseconds); 
END_IF 

IF Main.Errors.ProductHandlingErrors.Gantry_A.ProductLost[1] THEN 
Gantry_A_product_lost_section_1.Raise(Main.timestampNanoseconds); 
END_IF 

IF Main.Errors.ProductHandlingErrors.Gantry_A.ProductLost[2] THEN 
Gantry_A_product_lost_section_2.Raise(Main.timestampNanoseconds); 
END_IF 

IF Main.Errors.ProductHandlingErrors.Gantry_A.ProductLost[3] THEN 
Gantry_A_product_lost_section_3.Raise(Main.timestampNanoseconds); 
END_IF 

IF Main.Errors.ProductHandlingErrors.Gantry_A.ProductLost[4] THEN 
Gantry_A_product_lost_section_4.Raise(Main.timestampNanoseconds); 
END_IF 

IF Main.Errors.ProductHandlingErrors.Gantry_A.ProductLost[5] THEN 
Gantry_A_product_lost_section_5.Raise(Main.timestampNanoseconds); 
END_IF 

IF Main.Errors.ProductHandlingErrors.Gantry_A.ProductLost[6] THEN 
Gantry_A_product_lost_section_6.Raise(Main.timestampNanoseconds); 
END_IF 

IF Main.Errors.ProductHandlingErrors.Gantry_B.ProductLost[1] THEN 
Gantry_B_product_lost_section_1.Raise(Main.timestampNanoseconds); 
END_IF 

IF Main.Errors.ProductHandlingErrors.Gantry_B.ProductLost[2] THEN 
Gantry_B_product_lost_section_2.Raise(Main.timestampNanoseconds); 
END_IF 

IF Main.Errors.ProductHandlingErrors.Gantry_B.ProductLost[3] THEN 
Gantry_B_product_lost_section_3.Raise(Main.timestampNanoseconds); 
END_IF 

IF Main.Errors.ProductHandlingErrors.Gantry_B.ProductLost[4] THEN 
Gantry_B_product_lost_section_4.Raise(Main.timestampNanoseconds); 
END_IF 

IF Main.Errors.ProductHandlingErrors.Gantry_B.ProductLost[5] THEN 
Gantry_B_product_lost_section_5.Raise(Main.timestampNanoseconds); 
END_IF 

IF Main.Errors.ProductHandlingErrors.Gantry_B.ProductLost[6] THEN 
Gantry_B_product_lost_section_6.Raise(Main.timestampNanoseconds); 
END_IF 

IF Main.Errors.InMoldDryingErrors.ProductForming.SprayBar.PositionAtFrontError THEN 
Spraybar_not_in_front_rest_position.Raise(Main.timestampNanoseconds); 
END_IF 

IF Main.Errors.InMoldDryingErrors.ProductForming.SprayBar.PositionAtBackError THEN 
Spraybar_not_in_back_rest_position.Raise(Main.timestampNanoseconds); 
END_IF 

IF MAIN.EtherCatDiag.EtherCATLinkError THEN 
Ethercat_diagnosed_a_link_error.Raise(Main.timestampNanoseconds); 
END_IF 

IF MAIN.EtherCatDiag.EtherCATSlaveMissing THEN 
Ethercat_diagnosed_that_a_slave_is_missing.Raise(Main.timestampNanoseconds); 
END_IF 

IF MAIN.EtherCatDiag.EtherCATOPmode THEN 
Ethercat_diagnosed_a_non_OP_state.Raise(Main.timestampNanoseconds); 
END_IF 

IF MAIN.EtherCatDiag.EtherCATResetNeeded THEN 
Ethercat_diagnosed_that_a_ethercat_reset_is_needed.Raise(Main.timestampNanoseconds); 
END_IF 

IF Main.Errors.InMoldDryingErrors.TopMoldA.Hydraulic.SafePositionValveNotReached THEN 
TopMold_A_Safe_position_not_reached.Raise(Main.timestampNanoseconds); 
END_IF 

IF Main.Errors.InMoldDryingErrors.TopMoldB.Hydraulic.SafePositionValveNotReached THEN 
TopMold_B_Safe_position_not_reached.Raise(Main.timestampNanoseconds); 
END_IF 

IF Main.Errors.InMoldDryingErrors.TransferMold.HydraulicCilinder.SafePositionValveNotReached THEN 
Transfermold_Safe_position_not_reached.Raise(Main.timestampNanoseconds); 
END_IF 

IF Main.Errors.InMoldDryingErrors.TempDeviationToHighA[1] THEN 
Difference_in_temperature_too_high_top_bottommold_A_zone_1.Raise(Main.timestampNanoseconds); 
END_IF 

IF Main.Errors.InMoldDryingErrors.TempDeviationToHighA[2] THEN 
Difference_in_temperature_too_high_top_bottommold_A_zone_2.Raise(Main.timestampNanoseconds); 
END_IF 

IF Main.Errors.InMoldDryingErrors.TempDeviationToHighA[3] THEN 
Difference_in_temperature_too_high_top_bottommold_A_zone_3.Raise(Main.timestampNanoseconds); 
END_IF 

IF Main.Errors.InMoldDryingErrors.TempDeviationToHighA[4] THEN 
Difference_in_temperature_too_high_top_bottommold_A_zone_4.Raise(Main.timestampNanoseconds); 
END_IF 

IF Main.Errors.InMoldDryingErrors.TempDeviationToHighA[5] THEN 
Difference_in_temperature_too_high_top_bottommold_A_zone_5.Raise(Main.timestampNanoseconds); 
END_IF 

IF Main.Errors.InMoldDryingErrors.TempDeviationToHighA[6] THEN 
Difference_in_temperature_too_high_top_bottommold_A_zone_6.Raise(Main.timestampNanoseconds); 
END_IF 

IF Main.Errors.InMoldDryingErrors.TempDeviationToHighB[1] THEN 
Difference_in_temperature_too_high_top_bottommold_B_zone_1.Raise(Main.timestampNanoseconds); 
END_IF 

IF Main.Errors.InMoldDryingErrors.TempDeviationToHighB[2] THEN 
Difference_in_temperature_too_high_top_bottommold_B_zone_2.Raise(Main.timestampNanoseconds); 
END_IF 

IF Main.Errors.InMoldDryingErrors.TempDeviationToHighB[3] THEN 
Difference_in_temperature_too_high_top_bottommold_B_zone_3.Raise(Main.timestampNanoseconds); 
END_IF 

IF Main.Errors.InMoldDryingErrors.TempDeviationToHighB[4] THEN 
Difference_in_temperature_too_high_top_bottommold_B_zone_4.Raise(Main.timestampNanoseconds); 
END_IF 

IF Main.Errors.InMoldDryingErrors.TempDeviationToHighB[5] THEN 
Difference_in_temperature_too_high_top_bottommold_B_zone_5.Raise(Main.timestampNanoseconds); 
END_IF 

IF Main.Errors.InMoldDryingErrors.TempDeviationToHighB[6] THEN 
Difference_in_temperature_too_high_top_bottommold_B_zone_6.Raise(Main.timestampNanoseconds); 
END_IF 

IF Main.Errors.ProductHandlingErrors.Gantry_A.VerticalNCAxisError.exDriveAbsoluut THEN 
Gantry_A_Vertical_Drive_absoluut_error.Raise(Main.timestampNanoseconds); 
END_IF 

IF Main.Errors.ProductHandlingErrors.Gantry_A.VerticalNCAxisError.exDriveJog THEN 
Gantry_A_Vertical_Drive_Jog_error.Raise(Main.timestampNanoseconds); 
END_IF 

IF Main.Errors.ProductHandlingErrors.Gantry_A.VerticalNCAxisError.exDrivePower THEN 
Gantry_A_Vertical_Drive_power_error.Raise(Main.timestampNanoseconds); 
END_IF 

IF Main.Errors.ProductHandlingErrors.Gantry_A.VerticalNCAxisError.exDriveReset THEN 
Gantry_A_Vertical_Drive_reset.Raise(Main.timestampNanoseconds); 
END_IF 

IF Main.Errors.ProductHandlingErrors.Gantry_A.VerticalNCAxisError.exDriveStatus THEN 
Gantry_A_Vertical_Drive_status.Raise(Main.timestampNanoseconds); 
END_IF 

IF Main.Errors.ProductHandlingErrors.Gantry_A.VerticalNCAxisError.exDriveStop THEN 
Gantry_A_Vertical_Drive_stop_error.Raise(Main.timestampNanoseconds); 
END_IF 

IF Main.Errors.ProductHandlingErrors.Gantry_A.VerticalNCAxisError.exDriveVelocity THEN 
Gantry_A_Vertical_Drive_velocity_error.Raise(Main.timestampNanoseconds); 
END_IF 

IF Main.Errors.ProductHandlingErrors.Gantry_A.VerticalNCAxisError.exHome THEN 
Gantry_A_Vertical_Drive_home_error.Raise(Main.timestampNanoseconds); 
END_IF 

IF Main.Errors.ProductHandlingErrors.Gantry_A.VerticalNCAxisError.exLagError THEN 
Gantry_A_Vertical_Drive_lag_error.Raise(Main.timestampNanoseconds); 
END_IF 

IF Main.Errors.ProductHandlingErrors.Gantry_A.VerticalNCAxisError.exReadParameter THEN 
Gantry_A_Vertical_Drive_read_parameter_error.Raise(Main.timestampNanoseconds); 
END_IF 

IF Main.Errors.ProductHandlingErrors.Gantry_A.VerticalNCAxisError.exWriteParameter THEN 
Gantry_A_Vertical_Drive_write_parameter_error.Raise(Main.timestampNanoseconds); 
END_IF 

IF Main.Errors.ProductHandlingErrors.Gantry_B.VerticalNCAxisError.exDriveAbsoluut THEN 
Gantry_B_Vertical_Drive_absoluut_error.Raise(Main.timestampNanoseconds); 
END_IF 

IF Main.Errors.ProductHandlingErrors.Gantry_B.VerticalNCAxisError.exDriveJog THEN 
Gantry_B_Vertical_Drive_Jog_error.Raise(Main.timestampNanoseconds); 
END_IF 

IF Main.Errors.ProductHandlingErrors.Gantry_B.VerticalNCAxisError.exDrivePower THEN 
Gantry_B_Vertical_Drive_power_error.Raise(Main.timestampNanoseconds); 
END_IF 

IF Main.Errors.ProductHandlingErrors.Gantry_B.VerticalNCAxisError.exDriveReset THEN 
Gantry_B_Vertical_Drive_reset.Raise(Main.timestampNanoseconds); 
END_IF 

IF Main.Errors.ProductHandlingErrors.Gantry_B.VerticalNCAxisError.exDriveStatus THEN 
Gantry_B_Vertical_Drive_status.Raise(Main.timestampNanoseconds); 
END_IF 

IF Main.Errors.ProductHandlingErrors.Gantry_B.VerticalNCAxisError.exDriveStop THEN 
Gantry_B_Vertical_Drive_stop_error.Raise(Main.timestampNanoseconds); 
END_IF 

IF Main.Errors.ProductHandlingErrors.Gantry_B.VerticalNCAxisError.exDriveVelocity THEN 
Gantry_B_Vertical_Drive_velocity_error.Raise(Main.timestampNanoseconds); 
END_IF 

IF Main.Errors.ProductHandlingErrors.Gantry_B.VerticalNCAxisError.exHome THEN 
Gantry_B_Vertical_Drive_home_error.Raise(Main.timestampNanoseconds); 
END_IF 

IF Main.Errors.ProductHandlingErrors.Gantry_B.VerticalNCAxisError.exLagError THEN 
Gantry_B_Vertical_Drive_lag_error.Raise(Main.timestampNanoseconds); 
END_IF 

IF Main.Errors.ProductHandlingErrors.Gantry_B.VerticalNCAxisError.exReadParameter THEN 
Gantry_B_Vertical_Drive_read_parameter_error.Raise(Main.timestampNanoseconds); 
END_IF 

IF Main.Errors.ProductHandlingErrors.Gantry_B.VerticalNCAxisError.exWriteParameter THEN 
Gantry_B_Vertical_Drive_write_parameter_error.Raise(Main.timestampNanoseconds); 
END_IF 

IF Main.Errors.InMoldDryingErrors.BottomMoldB.HorizontalAxis.exDriveAbsoluut THEN 
Bottommold_B_Horizontal_Drive_absoluut_error.Raise(Main.timestampNanoseconds); 
END_IF 

IF Main.Errors.InMoldDryingErrors.BottomMoldB.HorizontalAxis.exDriveJog THEN 
Bottommold_B_Horizontal_Drive_Jog_error.Raise(Main.timestampNanoseconds); 
END_IF 

IF Main.Errors.InMoldDryingErrors.BottomMoldB.HorizontalAxis.exDrivePower THEN 
Bottommold_B_Horizontal_Drive_power_error.Raise(Main.timestampNanoseconds); 
END_IF 

IF Main.Errors.InMoldDryingErrors.BottomMoldB.HorizontalAxis.exDriveReset THEN 
Bottommold_B_Horizontal_Drive_reset.Raise(Main.timestampNanoseconds); 
END_IF 

IF Main.Errors.InMoldDryingErrors.BottomMoldB.HorizontalAxis.exDriveStatus THEN 
Bottommold_B_Horizontal_Drive_status.Raise(Main.timestampNanoseconds); 
END_IF 

IF Main.Errors.InMoldDryingErrors.BottomMoldB.HorizontalAxis.exDriveStop THEN 
Bottommold_B_Horizontal_Drive_stop_error.Raise(Main.timestampNanoseconds); 
END_IF 

IF Main.Errors.InMoldDryingErrors.BottomMoldB.HorizontalAxis.exDriveVelocity THEN 
Bottommold_B_Horizontal_Drive_velocity_error.Raise(Main.timestampNanoseconds); 
END_IF 

IF Main.Errors.InMoldDryingErrors.BottomMoldB.HorizontalAxis.exHome THEN 
Bottommold_B_Horizontal_Drive_home_error.Raise(Main.timestampNanoseconds); 
END_IF 

IF Main.Errors.InMoldDryingErrors.BottomMoldB.HorizontalAxis.exLagError THEN 
Bottommold_B_Horizontal_Drive_lag_error.Raise(Main.timestampNanoseconds); 
END_IF 

IF Main.Errors.InMoldDryingErrors.BottomMoldB.HorizontalAxis.exReadParameter THEN 
Bottommold_B_Horizontal_Drive_read_parameter_error.Raise(Main.timestampNanoseconds); 
END_IF 

IF Main.Errors.InMoldDryingErrors.BottomMoldB.HorizontalAxis.exWriteParameter THEN 
Bottommold_B_Horizontal_Drive_write_parameter_error.Raise(Main.timestampNanoseconds); 
END_IF 

IF Main.Errors.InMoldDryingErrors.BottomMoldA.HorizontalAxis.exDriveAbsoluut THEN 
Bottommold_A_Horizontal_Drive_absoluut_error.Raise(Main.timestampNanoseconds); 
END_IF 

IF Main.Errors.InMoldDryingErrors.BottomMoldA.HorizontalAxis.exDriveJog THEN 
Bottommold_A_Horizontal_Drive_Jog_error.Raise(Main.timestampNanoseconds); 
END_IF 

IF Main.Errors.InMoldDryingErrors.BottomMoldA.HorizontalAxis.exDrivePower THEN 
Bottommold_A_Horizontal_Drive_power_error.Raise(Main.timestampNanoseconds); 
END_IF 

IF Main.Errors.InMoldDryingErrors.BottomMoldA.HorizontalAxis.exDriveReset THEN 
Bottommold_A_Horizontal_Drive_reset.Raise(Main.timestampNanoseconds); 
END_IF 

IF Main.Errors.InMoldDryingErrors.BottomMoldA.HorizontalAxis.exDriveStatus THEN 
Bottommold_A_Horizontal_Drive_status.Raise(Main.timestampNanoseconds); 
END_IF 

IF Main.Errors.InMoldDryingErrors.BottomMoldA.HorizontalAxis.exDriveStop THEN 
Bottommold_A_Horizontal_Drive_stop_error.Raise(Main.timestampNanoseconds); 
END_IF 

IF Main.Errors.InMoldDryingErrors.BottomMoldA.HorizontalAxis.exDriveVelocity THEN 
Bottommold_A_Horizontal_Drive_velocity_error.Raise(Main.timestampNanoseconds); 
END_IF 

IF Main.Errors.InMoldDryingErrors.BottomMoldA.HorizontalAxis.exHome THEN 
Bottommold_A_Horizontal_Drive_home_error.Raise(Main.timestampNanoseconds); 
END_IF 

IF Main.Errors.InMoldDryingErrors.BottomMoldA.HorizontalAxis.exLagError THEN 
Bottommold_A_Horizontal_Drive_lag_error.Raise(Main.timestampNanoseconds); 
END_IF 

IF Main.Errors.InMoldDryingErrors.BottomMoldA.HorizontalAxis.exReadParameter THEN 
Bottommold_A_Horizontal_Drive_read_parameter_error.Raise(Main.timestampNanoseconds); 
END_IF 

IF Main.Errors.InMoldDryingErrors.BottomMoldA.HorizontalAxis.exWriteParameter THEN 
Bottommold_A_Horizontal_Drive_write_parameter_error.Raise(Main.timestampNanoseconds); 
END_IF
END_ACTION

END_PROGRAM

(* stored: Version 1.1.0.1, ProductVersion 3.1.4022.16
   POU HMI: Id {8c1b33ce-9977-4558-a527-7556af87d9de}, SpecialFunc None
   Action Error: Id {2a64f94b-fe6f-40aa-a153-b3f246d71ade} *)
